// TIA Portal V20 export
// export: Created 2025-09-14T10:55:00.0000000Z, ExportSetting WithDefaults
VAR_GLOBAL   // PLC tag table "Default tag table"
   RTU1_SF_RunFdbk AT %I0.0 : Bool;
   RTU1_SF_AirflowSw AT %I0.1 : Bool;
   RTU1_SF_VfdFault AT %I0.2 : Bool;
   RTU1_C_HighPressSw AT %I0.3 : Bool;
   RTU1_C_LowPressSw AT %I0.4 : Bool;
   RTU1_C_FreezeStat AT %I0.5 : Bool;
   RTU1_H_HighTempSw AT %I0.6 : Bool;
   RTU1_SYS_DirtyFilter AT %I0.7 : Bool;
   RTU1_SF_StartCmd AT %Q0.0 : Bool;
   RTU1_C_Comp1Cmd AT %Q0.1 : Bool;
   RTU1_H_Heat1Cmd AT %Q0.2 : Bool;
   RTU1_RAT_Temp AT %IW64 : Real;
   RTU1_OAT_Temp AT %IW66 : Real;
   RTU1_DAT_Temp AT %IW68 : Real;
   RTU1_SF_SpeedRef AT %QW64 : Real;
   RTU1_DMP_PosCmd AT %QW66 : Real;
END_VAR
